{attribute 'no_explicit_call' := 'do not call this POU directly'}
FUNCTION_BLOCK INTERNAL FB_RpcProxy IMPLEMENTS I_RpcProxy
VAR_INPUT
END_VAR
VAR_OUTPUT
END_VAR
VAR
	fbRpcSnappyVerify		: FB_RPC_Dynamic;
	sAmsNetID				: T_AmsNetID 			:= Param_TcHaxx_Snappy.cSnappyVerifyAmsNetID;
	nAmsPort				: T_AmsPort				:= Param_TcHaxx_Snappy.cSnappyVerifyPort;
	sInstancePathLocalField	: STRING				:= Param_TcHaxx_Snappy.cSnappyVerifyInstancePath;
	sSymbolLocalField		: STRING				:= Param_TcHaxx_Snappy.cSnappyVerifySymbol;
	bIsConfiguredField		: BOOL					:= FALSE;
	stVerificationResult	: ST_VerificationResult;
END_VAR

PROPERTY bIsConfigured : BOOL
GET
bIsConfigured := bIsConfiguredField;
END_GET
END_PROPERTY

METHOD GetVerificationResult : HRESULT
VAR_OUTPUT
	stResult : ST_VerificationResult;
END_VAR

VAR
	stAdsStatus	: TcHaxx.ST_AdsStatus;
END_VAR
GetVerificationResult := S_PENDING;

stAdsStatus := THIS^.fbRpcSnappyVerify.Invoke();

IF NOT stAdsStatus.bBusy AND NOT stAdsStatus.bError THEN
	GetVerificationResult := S_OK;
	stResult := stVerificationResult;
	RETURN;
ELSIF stAdsStatus.bError THEN
	GetVerificationResult := TO_DINT(stAdsStatus.nError);
	RETURN;
END_IF
END_METHOD

METHOD Verify : HRESULT
VAR_INPUT CONSTANT
	sToVerify	: REFERENCE TO T_VerifyContent;
END_VAR
VAR
	hr			: HRESULT;
	stAdsStatus	: TcHaxx.ST_AdsStatus;
END_VAR
IF NOT bIsConfiguredField THEN
	hr := fbRpcSnappyVerify.Configure()
			.WithAmsNetId(sAmsNetId:= THIS^.sAmsNetID)
			.WithAmsPort(nAmsPort:= THIS^.nAmsPort)
			.WithSymbolPath(sInstancePath:= THIS^.sInstancePathLocalField, sSymbol:= THIS^.sSymbolLocalField)
			.Build();
	bIsConfiguredField := SUCCEEDED(hr);
END_IF;

IF NOT bIsConfigured THEN
	Verify := E_HRESULTAdsErr.NOTINIT;
	RETURN;
END_IF

stAdsStatus := fbRpcSnappyVerify.VarInput(anyArg:= sToVerify).ReturnValue(anyRetVal:= stVerificationResult).Invoke();
IF stAdsStatus.bError THEN
	Verify := TO_DINT(stAdsStatus.nError);
	RETURN;
END_IF

Verify := S_PENDING;
END_METHOD

END_FUNCTION_BLOCK

(* stored: Version 1.1.0.1, ProductVersion 3.1.4024.12
   POU FB_RpcProxy: Id {f9e7075c-2104-427f-9a7e-5e84f1a64890}, SpecialFunc None
   Property bIsConfigured: Id {66d99f6c-2f7b-4335-8601-3cb01d592de5}
   Get Get: Id {b1f9bb6c-7f5e-474a-9938-247984a86174}
   Method GetVerificationResult: Id {a7278404-bd08-4a34-9891-a82b07ef5350}
   Method Verify: Id {1f2ed438-c0f1-406f-9917-7be1f3353347} *)
